FUNCTION_BLOCK ADD_UINT (* IEC 61131-3 UINT Addition *)
  (* Standard: 61131-3 *)
  (* Version 0.0, 2004-12-15, JHC, Rockwell Automation, Converted from SRC format. *)
  (* Compiler header: package fb.rt.plc.math; *)
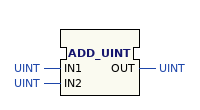
  VAR_INPUT
    IN1 : UINT; (* Augend *)
    IN2 : UINT; (* Addend *)
  END_VAR
  VAR_OUTPUT
    OUT : UINT; (* Sum *)
  END_VAR
END_FUNCTION_BLOCK
